// TIA Portal V20 export
ORGANIZATION_BLOCK "Startup"   // OB1050, LAD, Startup
TITLE = "Complete Restart"
AUTHOR : ERsystem_FA2_DH. Kim
// stored: AutoNumber false, IsIECCheckEnabled true, Namespace Unit1.Em5, SetENOAutomatically false
   VAR_INPUT
      LostRetentive : Bool;   // True if retentive data are lost
      LostRTC : Bool;   // True if date and time are lost
   END_VAR
BEGIN

REGION Network 1 (SCL): Build the Absolut Reference Designator
   // Set the Absoult Reference Designator in the Config DB
   IF LEN(IN := "Unit1.Em5.Config".em.referenceDesignator.parent) <> 0 THEN
     "Unit1.Em5.Config".em.referenceDesignator.combined := CONCAT_WSTRING(IN1 := "Unit1.Em5.Config".em.referenceDesignator.parent, IN2 := WSTRING#'.', IN3 := "Unit1.Em5.Config".em.referenceDesignator.relative);
   ELSE
     "Unit1.Em5.Config".em.referenceDesignator.combined := "Unit1.Em5.Config".em.referenceDesignator.relative;
   END_IF;
END_REGION

REGION Network 2 (SCL): Assign axes data
   //Assign axes
   "Unit1.Em5.Config".axis[1] := "BA040AZSCDR7_CathodeMainPnp1AxisX";
   "Unit1.Em5.Config".axis[2] := "BA040AZSCDR8_CathodeMainPnp2AxisX";
   "Unit1.Em5.Config".axis[3] := "BA040AZSCDR9_CathodeMainPnp1AxisY";
   "Unit1.Em5.Config".axis[4] := "BA040AZSCDR10_CathodeMainPnp1AxisZ";
   "Unit1.Em5.Config".axis[5] := "BA040AZSCDR13_CathodeMainPnp2AxisZ";
   "Unit1.Em5.Config".axis[6] := "BA040AZSCDR18_CathodeAlignTableAxisX";
   "Unit1.Em5.Config".axis[7] := "BA040AZSCDR19_CathodeAlignTableAxisY1";
   "Unit1.Em5.Config".axis[8] := "BA040AZSCDR20_CathodeAlignTableAxisY2";

   // Config.cam[1] := _.BA030AZSCDR5_cathodeMainPnp1AxisXCamMain;
   // Config.cam[2] := _.BA030AZSCDR6_cathodeMainPnp2AxisXCamMain;
   // Config.cam[3] := _.BA030AZSCDR12_cathodeMainPnp1AxisZCamMain;
   // Config.cam[4] := _.BA030AZSCDR14_cathodeMainPnp2AxisZCamMain;

   "Unit1.Em5.Config".outputCam[1] := "CathodePnP1XFwd";
   "Unit1.Em5.Config".outputCam[2] := "CathodePnP1XBwd";
   "Unit1.Em5.Config".outputCam[3] := "CathodePnP2XFwd";
   "Unit1.Em5.Config".outputCam[4] := "CathodePnP2XBwd";
   "Unit1.Em5.Config".outputCam[5] := "CathodePnPZ1Down1";
   "Unit1.Em5.Config".outputCam[6] := "CathodePnPZ1Up1";
   "Unit1.Em5.Config".outputCam[7] := "CathodePnPZ2Down1";
   "Unit1.Em5.Config".outputCam[8] := "CathodePnPZ2Up1";
   "Unit1.Em5.Config".outputCam[9] := "CathodePnPZ1Down2";
   "Unit1.Em5.Config".outputCam[10] := "CathodePnPZ1Up2";
   "Unit1.Em5.Config".outputCam[11] := "CathodePnPZ2Down2";
   "Unit1.Em5.Config".outputCam[12] := "CathodePnPZ2Up2";
   "Unit1.Em5.Config".outputCam[13] := "CathodePnPZ1SuctionOn";
   "Unit1.Em5.Config".outputCam[14] := "CathodePnPZ1SuctionOff";
   "Unit1.Em5.Config".outputCam[15] := "CathodePnPZ1ReelCutBlow";
   "Unit1.Em5.Config".outputCam[16] := "CathodePnPZ2SuctionOn";
   "Unit1.Em5.Config".outputCam[17] := "CathodePnPZ2SuctionOff";
   "Unit1.Em5.Config".outputCam[18] := "CathodeAlignSuctionOn";
   "Unit1.Em5.Config".outputCam[19] := "CathodeAlignSuctionOff";

   // Assign configuration data of axis

   // FB Enable
   "Unit1.Em5.HmiInterface".cmCathodeMainPnP1AxisX.commands.enableMasterControl := TRUE;
   "Unit1.Em5.HmiInterface".cmCathodeMainPnP1AxisY.commands.enableMasterControl := TRUE;
   "Unit1.Em5.HmiInterface".cmCathodeMainPnP1AxisZ.commands.enableMasterControl := TRUE;
   "Unit1.Em5.HmiInterface".cmCathodeMainPnP2AxisX.commands.enableMasterControl := TRUE;
   "Unit1.Em5.HmiInterface".cmCathodeMainPnP2AxisZ.commands.enableMasterControl := TRUE;
   "Unit1.Em5.HmiInterface".cmCathodeAlignTableAxisX.commands.enableMasterControl := TRUE;
   "Unit1.Em5.HmiInterface".cmCathodeAlignTableAxisY1.commands.enableMasterControl := TRUE;
   "Unit1.Em5.HmiInterface".cmCathodeAlignTableAxisY2.commands.enableMasterControl := TRUE;

   // Axis 1 BA030AZSCDR6_CathodeMainPnp1AxisX
   "Unit1.Em5.HmiInterface".cmCathodeMainPnP1AxisX.commandConfiguration.jog.velocity := 10.0;
   "Unit1.Em5.HmiInterface".cmCathodeMainPnP1AxisX.commandConfiguration.jog.acceleration := 100.0;
   "Unit1.Em5.HmiInterface".cmCathodeMainPnP1AxisX.commandConfiguration.jog.deceleration := 100.0;
   "Unit1.Em5.HmiInterface".cmCathodeMainPnP1AxisX.commandConfiguration.moveVelocity.velocity := 10.0;
   "Unit1.Em5.HmiInterface".cmCathodeMainPnP1AxisX.commandConfiguration.moveVelocity.acceleration := 100.0;
   "Unit1.Em5.HmiInterface".cmCathodeMainPnP1AxisX.commandConfiguration.moveVelocity.deceleration := 100.0;
   "Unit1.Em5.HmiInterface".cmCathodeMainPnP1AxisX.commandConfiguration.posRelative.velocity := 10.0;
   "Unit1.Em5.HmiInterface".cmCathodeMainPnP1AxisX.commandConfiguration.posRelative.acceleration := 100.0;
   "Unit1.Em5.HmiInterface".cmCathodeMainPnP1AxisX.commandConfiguration.posRelative.deceleration := 100.0;
   "Unit1.Em5.HmiInterface".cmCathodeMainPnP1AxisX.configuration.setPositions[0].name := 'reelCutConveyerPos';
   "Unit1.Em5.HmiInterface".cmCathodeMainPnP1AxisX.configuration.setPositions[1].name := 'alignTablePos';

   // Axis 2 BA030AZSCDR8_CathodeMainPnp2AxisX
   "Unit1.Em5.HmiInterface".cmCathodeMainPnP2AxisX.commandConfiguration.jog.velocity := 10.0;
   "Unit1.Em5.HmiInterface".cmCathodeMainPnP2AxisX.commandConfiguration.jog.acceleration := 100.0;
   "Unit1.Em5.HmiInterface".cmCathodeMainPnP2AxisX.commandConfiguration.jog.deceleration := 100.0;
   "Unit1.Em5.HmiInterface".cmCathodeMainPnP2AxisX.commandConfiguration.moveVelocity.velocity := 10.0;
   "Unit1.Em5.HmiInterface".cmCathodeMainPnP2AxisX.commandConfiguration.moveVelocity.acceleration := 100.0;
   "Unit1.Em5.HmiInterface".cmCathodeMainPnP2AxisX.commandConfiguration.moveVelocity.deceleration := 100.0;
   "Unit1.Em5.HmiInterface".cmCathodeMainPnP2AxisX.commandConfiguration.posRelative.velocity := 10.0;
   "Unit1.Em5.HmiInterface".cmCathodeMainPnP2AxisX.commandConfiguration.posRelative.acceleration := 100.0;
   "Unit1.Em5.HmiInterface".cmCathodeMainPnP2AxisX.commandConfiguration.posRelative.deceleration := 100.0;
   "Unit1.Em5.HmiInterface".cmCathodeMainPnP2AxisX.configuration.setPositions[0].name := 'alignTablePos';
   "Unit1.Em5.HmiInterface".cmCathodeMainPnP2AxisX.configuration.setPositions[1].name := 'stackTablePos';

   // Axis3 BA030AZSCDR11_CathodeMainPnp1AxisY
   "Unit1.Em5.HmiInterface".cmCathodeMainPnP1AxisY.commandConfiguration.jog.velocity := 10.0;
   "Unit1.Em5.HmiInterface".cmCathodeMainPnP1AxisY.commandConfiguration.jog.acceleration := 100.0;
   "Unit1.Em5.HmiInterface".cmCathodeMainPnP1AxisY.commandConfiguration.jog.deceleration := 100.0;
   "Unit1.Em5.HmiInterface".cmCathodeMainPnP1AxisY.commandConfiguration.moveVelocity.velocity := 10.0;
   "Unit1.Em5.HmiInterface".cmCathodeMainPnP1AxisY.commandConfiguration.moveVelocity.acceleration := 100.0;
   "Unit1.Em5.HmiInterface".cmCathodeMainPnP1AxisY.commandConfiguration.moveVelocity.deceleration := 100.0;
   "Unit1.Em5.HmiInterface".cmCathodeMainPnP1AxisY.commandConfiguration.posRelative.velocity := 10.0;
   "Unit1.Em5.HmiInterface".cmCathodeMainPnP1AxisY.commandConfiguration.posRelative.acceleration := 100.0;
   "Unit1.Em5.HmiInterface".cmCathodeMainPnP1AxisY.commandConfiguration.posRelative.deceleration := 100.0;
   "Unit1.Em5.HmiInterface".cmCathodeMainPnP1AxisY.configuration.setPositions[0].name := 'waitPos';

   // Axis 4 BA030AZSCDR12_CathodeMainPnp1AxisZ
   "Unit1.Em5.HmiInterface".cmCathodeMainPnP1AxisZ.commandConfiguration.jog.velocity := 10.0;
   "Unit1.Em5.HmiInterface".cmCathodeMainPnP1AxisZ.commandConfiguration.jog.acceleration := 100.0;
   "Unit1.Em5.HmiInterface".cmCathodeMainPnP1AxisZ.commandConfiguration.jog.deceleration := 100.0;
   "Unit1.Em5.HmiInterface".cmCathodeMainPnP1AxisZ.commandConfiguration.moveVelocity.velocity := 10.0;
   "Unit1.Em5.HmiInterface".cmCathodeMainPnP1AxisZ.commandConfiguration.moveVelocity.acceleration := 100.0;
   "Unit1.Em5.HmiInterface".cmCathodeMainPnP1AxisZ.commandConfiguration.moveVelocity.deceleration := 100.0;
   "Unit1.Em5.HmiInterface".cmCathodeMainPnP1AxisZ.commandConfiguration.posRelative.velocity := 10.0;
   "Unit1.Em5.HmiInterface".cmCathodeMainPnP1AxisZ.commandConfiguration.posRelative.acceleration := 100.0;
   "Unit1.Em5.HmiInterface".cmCathodeMainPnP1AxisZ.commandConfiguration.posRelative.deceleration := 100.0;
   "Unit1.Em5.HmiInterface".cmCathodeMainPnP1AxisZ.configuration.setPositions[0].name := 'upPos';
   "Unit1.Em5.HmiInterface".cmCathodeMainPnP1AxisZ.configuration.setPositions[1].name := 'reelCutConveyerDownPos';
   "Unit1.Em5.HmiInterface".cmCathodeMainPnP1AxisZ.configuration.setPositions[2].name := 'ailgnTableDownPos';

   // Axis 5 BA030AZSCDR14_CathodeMainPnp2AxisZ
   "Unit1.Em5.HmiInterface".cmCathodeMainPnP2AxisZ.commandConfiguration.jog.velocity := 10.0;
   "Unit1.Em5.HmiInterface".cmCathodeMainPnP2AxisZ.commandConfiguration.jog.acceleration := 100.0;
   "Unit1.Em5.HmiInterface".cmCathodeMainPnP2AxisZ.commandConfiguration.jog.deceleration := 100.0;
   "Unit1.Em5.HmiInterface".cmCathodeMainPnP2AxisZ.commandConfiguration.moveVelocity.velocity := 10.0;
   "Unit1.Em5.HmiInterface".cmCathodeMainPnP2AxisZ.commandConfiguration.moveVelocity.acceleration := 100.0;
   "Unit1.Em5.HmiInterface".cmCathodeMainPnP2AxisZ.commandConfiguration.moveVelocity.deceleration := 100.0;
   "Unit1.Em5.HmiInterface".cmCathodeMainPnP2AxisZ.commandConfiguration.posRelative.velocity := 10.0;
   "Unit1.Em5.HmiInterface".cmCathodeMainPnP2AxisZ.commandConfiguration.posRelative.acceleration := 100.0;
   "Unit1.Em5.HmiInterface".cmCathodeMainPnP2AxisZ.commandConfiguration.posRelative.deceleration := 100.0;
   "Unit1.Em5.HmiInterface".cmCathodeMainPnP2AxisZ.configuration.setPositions[0].name := 'upPos';
   "Unit1.Em5.HmiInterface".cmCathodeMainPnP2AxisZ.configuration.setPositions[1].name := 'ailgnTableDownPos';
   "Unit1.Em5.HmiInterface".cmCathodeMainPnP2AxisZ.configuration.setPositions[2].name := 'stackTableDownPos';

   // Axis 6 BA030AZSCDR18_CathodeAlignTableAxisX
   "Unit1.Em5.HmiInterface".cmCathodeAlignTableAxisX.commandConfiguration.jog.velocity := 10.0;
   "Unit1.Em5.HmiInterface".cmCathodeAlignTableAxisX.commandConfiguration.jog.acceleration := 100.0;
   "Unit1.Em5.HmiInterface".cmCathodeAlignTableAxisX.commandConfiguration.jog.deceleration := 100.0;
   "Unit1.Em5.HmiInterface".cmCathodeAlignTableAxisX.commandConfiguration.moveVelocity.velocity := 10.0;
   "Unit1.Em5.HmiInterface".cmCathodeAlignTableAxisX.commandConfiguration.moveVelocity.acceleration := 100.0;
   "Unit1.Em5.HmiInterface".cmCathodeAlignTableAxisX.commandConfiguration.moveVelocity.deceleration := 100.0;
   "Unit1.Em5.HmiInterface".cmCathodeAlignTableAxisX.commandConfiguration.posRelative.velocity := 10.0;
   "Unit1.Em5.HmiInterface".cmCathodeAlignTableAxisX.commandConfiguration.posRelative.acceleration := 100.0;
   "Unit1.Em5.HmiInterface".cmCathodeAlignTableAxisX.commandConfiguration.posRelative.deceleration := 100.0;
   "Unit1.Em5.HmiInterface".cmCathodeAlignTableAxisX.configuration.setPositions[0].name := 'waitPos';
   "Unit1.Em5.HmiInterface".cmCathodeAlignTableAxisX.configuration.setPositions[1].name := 'adjustPos';

   // Axis 7 BA030AZSCDR19_CathodeAlignTableAxisY1
   "Unit1.Em5.HmiInterface".cmCathodeAlignTableAxisY1.commandConfiguration.jog.velocity := 10.0;
   "Unit1.Em5.HmiInterface".cmCathodeAlignTableAxisY1.commandConfiguration.jog.acceleration := 100.0;
   "Unit1.Em5.HmiInterface".cmCathodeAlignTableAxisY1.commandConfiguration.jog.deceleration := 100.0;
   "Unit1.Em5.HmiInterface".cmCathodeAlignTableAxisY1.commandConfiguration.moveVelocity.velocity := 10.0;
   "Unit1.Em5.HmiInterface".cmCathodeAlignTableAxisY1.commandConfiguration.moveVelocity.acceleration := 100.0;
   "Unit1.Em5.HmiInterface".cmCathodeAlignTableAxisY1.commandConfiguration.moveVelocity.deceleration := 100.0;
   "Unit1.Em5.HmiInterface".cmCathodeAlignTableAxisY1.commandConfiguration.posRelative.velocity := 10.0;
   "Unit1.Em5.HmiInterface".cmCathodeAlignTableAxisY1.commandConfiguration.posRelative.acceleration := 100.0;
   "Unit1.Em5.HmiInterface".cmCathodeAlignTableAxisY1.commandConfiguration.posRelative.deceleration := 100.0;
   "Unit1.Em5.HmiInterface".cmCathodeAlignTableAxisY1.configuration.setPositions[0].name := 'waitPos';
   "Unit1.Em5.HmiInterface".cmCathodeAlignTableAxisY1.configuration.setPositions[1].name := 'adjustPos';

   // Axis 8 BA030AZSCDR20_CathodeAlignTableAxisY2
   "Unit1.Em5.HmiInterface".cmCathodeAlignTableAxisY2.commandConfiguration.jog.velocity := 10.0;
   "Unit1.Em5.HmiInterface".cmCathodeAlignTableAxisY2.commandConfiguration.jog.acceleration := 100.0;
   "Unit1.Em5.HmiInterface".cmCathodeAlignTableAxisY2.commandConfiguration.jog.deceleration := 100.0;
   "Unit1.Em5.HmiInterface".cmCathodeAlignTableAxisY2.commandConfiguration.moveVelocity.velocity := 10.0;
   "Unit1.Em5.HmiInterface".cmCathodeAlignTableAxisY2.commandConfiguration.moveVelocity.acceleration := 100.0;
   "Unit1.Em5.HmiInterface".cmCathodeAlignTableAxisY2.commandConfiguration.moveVelocity.deceleration := 100.0;
   "Unit1.Em5.HmiInterface".cmCathodeAlignTableAxisY2.commandConfiguration.posRelative.velocity := 10.0;
   "Unit1.Em5.HmiInterface".cmCathodeAlignTableAxisY2.commandConfiguration.posRelative.acceleration := 100.0;
   "Unit1.Em5.HmiInterface".cmCathodeAlignTableAxisY2.commandConfiguration.posRelative.deceleration := 100.0;
   "Unit1.Em5.HmiInterface".cmCathodeAlignTableAxisY2.configuration.setPositions[0].name := 'waitPos';
   "Unit1.Em5.HmiInterface".cmCathodeAlignTableAxisY2.configuration.setPositions[1].name := 'adjustPos';
END_REGION

REGION Network 3 (SCL): Assign TwoWayActuator data
   //Assign Configuration data of TwoWayActuator

   //cmCathodeMainPnP1RotaryCwCcw
   "Unit1.Em5.Config".cmCathodeMainPnP1RotaryCwCcw.referenceDesignator := WSTRING#'MainPnP1RotaryCwCcw';
   "Unit1.Em5.Config".cmCathodeMainPnP1RotaryCwCcw.disableFeedbackHomePos := FALSE;
   "Unit1.Em5.Config".cmCathodeMainPnP1RotaryCwCcw.disableFeedbackWorkPos := FALSE;
   "Unit1.Em5.HmiInterface".cmCathodeMainPnP1RotaryCwCcw.configuration.referenceDesignator := WSTRING#'MainPnP1RotaryCwCcw';
   "Unit1.Em5.HmiInterface".cmCathodeMainPnP1RotaryCwCcw.configuration.disableFeedbackHomePos := FALSE;
   "Unit1.Em5.HmiInterface".cmCathodeMainPnP1RotaryCwCcw.configuration.disableFeedbackWorkPos := FALSE;

   //cmCathodeMainPnP1SuctionPlateVacuum
   "Unit1.Em5.Config".cmCathodeMainPnP1SuctionPlateVacuum.referenceDesignator := WSTRING#'MainPnP1Vacuum';
   "Unit1.Em5.Config".cmCathodeMainPnP1SuctionPlateVacuum.disableFeedbackHomePos := FALSE;
   "Unit1.Em5.Config".cmCathodeMainPnP1SuctionPlateVacuum.disableFeedbackWorkPos := FALSE;
   "Unit1.Em5.HmiInterface".cmCathodeMainPnP1SuctionPlateVacuum.configuration.referenceDesignator := WSTRING#'MainPnP1Vacuum';
   "Unit1.Em5.HmiInterface".cmCathodeMainPnP1SuctionPlateVacuum.configuration.disableFeedbackHomePos := FALSE;
   "Unit1.Em5.HmiInterface".cmCathodeMainPnP1SuctionPlateVacuum.configuration.disableFeedbackWorkPos := FALSE;

   //cmCathodeMainPnP2SuctionPlateVacuum
   "Unit1.Em5.Config".cmCathodeMainPnP2SuctionPlateVacuum.referenceDesignator := WSTRING#'MainPnP2Vacuum';
   "Unit1.Em5.Config".cmCathodeMainPnP2SuctionPlateVacuum.disableFeedbackHomePos := FALSE;
   "Unit1.Em5.Config".cmCathodeMainPnP2SuctionPlateVacuum.disableFeedbackWorkPos := FALSE;
   "Unit1.Em5.HmiInterface".cmCathodeMainPnP2SuctionPlateVacuum.configuration.referenceDesignator := WSTRING#'MainPnP2Vacuum';
   "Unit1.Em5.HmiInterface".cmCathodeMainPnP2SuctionPlateVacuum.configuration.disableFeedbackHomePos := FALSE;
   "Unit1.Em5.HmiInterface".cmCathodeMainPnP2SuctionPlateVacuum.configuration.disableFeedbackWorkPos := FALSE;

   //cmCathodeAlignTableSuctionPlateVacuum
   "Unit1.Em5.Config".cmCathodeAlignTableSuctionPlateVacuum.referenceDesignator := WSTRING#'AlignTableVaccum';
   "Unit1.Em5.Config".cmCathodeAlignTableSuctionPlateVacuum.disableFeedbackHomePos := FALSE;
   "Unit1.Em5.Config".cmCathodeAlignTableSuctionPlateVacuum.disableFeedbackWorkPos := FALSE;
   "Unit1.Em5.HmiInterface".cmCathodeAlignTableSuctionPlateVacuum.configuration.referenceDesignator := WSTRING#'AlignTableVaccum';
   "Unit1.Em5.HmiInterface".cmCathodeAlignTableSuctionPlateVacuum.configuration.disableFeedbackHomePos := FALSE;
   "Unit1.Em5.HmiInterface".cmCathodeAlignTableSuctionPlateVacuum.configuration.disableFeedbackWorkPos := FALSE;

   //cmCathodeGlassCleaning
   "Unit1.Em5.Config".cmCathodeGlassCleaning.referenceDesignator := WSTRING#'GlassCleaning';
   "Unit1.Em5.Config".cmCathodeGlassCleaning.disableFeedbackHomePos := TRUE;
   "Unit1.Em5.Config".cmCathodeGlassCleaning.disableFeedbackWorkPos := TRUE;
   "Unit1.Em5.HmiInterface".cmCathodeGlassCleaning.configuration.referenceDesignator := WSTRING#'GlassCleaning';
   "Unit1.Em5.HmiInterface".cmCathodeGlassCleaning.configuration.disableFeedbackHomePos := TRUE;
   "Unit1.Em5.HmiInterface".cmCathodeGlassCleaning.configuration.disableFeedbackWorkPos := TRUE;

   //cmCathodeNgPnpUpDown
   "Unit1.Em5.Config".cmCathodeNgPnpUpDown.referenceDesignator := WSTRING#'NgPnpUpDown';
   "Unit1.Em5.Config".cmCathodeNgPnpUpDown.disableFeedbackHomePos := FALSE;
   "Unit1.Em5.Config".cmCathodeNgPnpUpDown.disableFeedbackWorkPos := FALSE;
   "Unit1.Em5.HmiInterface".cmCathodeNgPnpUpDown.configuration.referenceDesignator := WSTRING#'NgPnpUpDown';
   "Unit1.Em5.HmiInterface".cmCathodeNgPnpUpDown.configuration.disableFeedbackHomePos := FALSE;
   "Unit1.Em5.HmiInterface".cmCathodeNgPnpUpDown.configuration.disableFeedbackWorkPos := FALSE;

   //cmCathodeNgPnp1stFwdBwd
   "Unit1.Em5.Config".cmCathodeNgPnp1stFwdBwd.referenceDesignator := WSTRING#'NgPnp1stFwdBwd';
   "Unit1.Em5.Config".cmCathodeNgPnp1stFwdBwd.disableFeedbackHomePos := FALSE;
   "Unit1.Em5.Config".cmCathodeNgPnp1stFwdBwd.disableFeedbackWorkPos := FALSE;
   "Unit1.Em5.HmiInterface".cmCathodeNgPnp1stFwdBwd.configuration.referenceDesignator := WSTRING#'NgPnp1stFwdBwd';
   "Unit1.Em5.HmiInterface".cmCathodeNgPnp1stFwdBwd.configuration.disableFeedbackHomePos := FALSE;
   "Unit1.Em5.HmiInterface".cmCathodeNgPnp1stFwdBwd.configuration.disableFeedbackWorkPos := FALSE;

   //cmCathodeNgPnp2ndFwdBwd
   "Unit1.Em5.Config".cmCathodeNgPnp2ndFwdBwd.referenceDesignator := WSTRING#'NgPnp2ndFwdBwd';
   "Unit1.Em5.Config".cmCathodeNgPnp2ndFwdBwd.disableFeedbackHomePos := FALSE;
   "Unit1.Em5.Config".cmCathodeNgPnp2ndFwdBwd.disableFeedbackWorkPos := FALSE;
   "Unit1.Em5.HmiInterface".cmCathodeNgPnp2ndFwdBwd.configuration.referenceDesignator := WSTRING#'NgPnp2ndFwdBwd';
   "Unit1.Em5.HmiInterface".cmCathodeNgPnp2ndFwdBwd.configuration.disableFeedbackHomePos := FALSE;
   "Unit1.Em5.HmiInterface".cmCathodeNgPnp2ndFwdBwd.configuration.disableFeedbackWorkPos := FALSE;

   //cmCathodeMaintenanceMovingFixFrontRearFwdBwd
   "Unit1.Em5.Config".cmCathodeMaintenanceMovingFixFrontRearFwdBwd.referenceDesignator := WSTRING#'MaintenanceFix';
   "Unit1.Em5.Config".cmCathodeMaintenanceMovingFixFrontRearFwdBwd.disableFeedbackHomePos := FALSE;
   "Unit1.Em5.Config".cmCathodeMaintenanceMovingFixFrontRearFwdBwd.disableFeedbackWorkPos := FALSE;
   "Unit1.Em5.HmiInterface".cmCathodeMaintenanceMovingFixFrontRearFwdBwd.configuration.referenceDesignator := WSTRING#'MaintenanceFix';
   "Unit1.Em5.HmiInterface".cmCathodeMaintenanceMovingFixFrontRearFwdBwd.configuration.disableFeedbackHomePos := FALSE;
   "Unit1.Em5.HmiInterface".cmCathodeMaintenanceMovingFixFrontRearFwdBwd.configuration.disableFeedbackWorkPos := FALSE;

   //cmCathodeNgBoxLiftUpDown
   "Unit1.Em5.Config".cmCathodeNgBoxLiftUpDown.referenceDesignator := WSTRING#'NgBoxLiftUpDown';
   "Unit1.Em5.Config".cmCathodeNgBoxLiftUpDown.disableFeedbackHomePos := FALSE;
   "Unit1.Em5.Config".cmCathodeNgBoxLiftUpDown.disableFeedbackWorkPos := FALSE;
   "Unit1.Em5.HmiInterface".cmCathodeNgBoxLiftUpDown.configuration.referenceDesignator := WSTRING#'NgBoxLiftUpDown';
   "Unit1.Em5.HmiInterface".cmCathodeNgBoxLiftUpDown.configuration.disableFeedbackHomePos := FALSE;
   "Unit1.Em5.HmiInterface".cmCathodeNgBoxLiftUpDown.configuration.disableFeedbackWorkPos := FALSE;

   //cmCathodeNgBoxLockUpDown
   "Unit1.Em5.Config".cmCathodeNgBoxLockUpDown.referenceDesignator := WSTRING#'NgBoxLockUpDown';
   "Unit1.Em5.Config".cmCathodeNgBoxLockUpDown.disableFeedbackHomePos := FALSE;
   "Unit1.Em5.Config".cmCathodeNgBoxLockUpDown.disableFeedbackWorkPos := FALSE;
   "Unit1.Em5.HmiInterface".cmCathodeNgBoxLockUpDown.configuration.referenceDesignator := WSTRING#'NgBoxLockUpDown';
   "Unit1.Em5.HmiInterface".cmCathodeNgBoxLockUpDown.configuration.disableFeedbackHomePos := FALSE;
   "Unit1.Em5.HmiInterface".cmCathodeNgBoxLockUpDown.configuration.disableFeedbackWorkPos := FALSE;

   //cmCathodeNgPnpVaccum
   "Unit1.Em5.Config".cmCathodeNgPnpVaccum.referenceDesignator := WSTRING#'NgPnpVaccum';
   "Unit1.Em5.Config".cmCathodeNgPnpVaccum.disableFeedbackHomePos := FALSE;
   "Unit1.Em5.Config".cmCathodeNgPnpVaccum.disableFeedbackWorkPos := FALSE;
   "Unit1.Em5.HmiInterface".cmCathodeNgPnpVaccum.configuration.referenceDesignator := WSTRING#'NgPnpVaccum';
   "Unit1.Em5.HmiInterface".cmCathodeNgPnpVaccum.configuration.disableFeedbackHomePos := FALSE;
   "Unit1.Em5.HmiInterface".cmCathodeNgPnpVaccum.configuration.disableFeedbackWorkPos := FALSE;

   //cmCathodeConveyorCoverFwdBwd
   "Unit1.Em5.Config".cmCathodeConveyorCoverFwdBwd.referenceDesignator := WSTRING#'ConveyorCoverFwdBwd';
   "Unit1.Em5.Config".cmCathodeConveyorCoverFwdBwd.disableFeedbackHomePos := FALSE;
   "Unit1.Em5.Config".cmCathodeConveyorCoverFwdBwd.disableFeedbackWorkPos := FALSE;
   "Unit1.Em5.HmiInterface".cmCathodeConveyorCoverFwdBwd.configuration.referenceDesignator := WSTRING#'ConveyorCoverFwdBwd';
   "Unit1.Em5.HmiInterface".cmCathodeConveyorCoverFwdBwd.configuration.disableFeedbackHomePos := FALSE;
   "Unit1.Em5.HmiInterface".cmCathodeConveyorCoverFwdBwd.configuration.disableFeedbackWorkPos := FALSE;

   //cmCathodeConveyorPickUpBlower
   "Unit1.Em5.Config".cmCathodeConveyorPickUpBlower.referenceDesignator := WSTRING#'ConveyorPickUpBlower';
   "Unit1.Em5.Config".cmCathodeConveyorPickUpBlower.disableFeedbackHomePos := TRUE;
   "Unit1.Em5.Config".cmCathodeConveyorPickUpBlower.disableFeedbackWorkPos := TRUE;
   "Unit1.Em5.HmiInterface".cmCathodeConveyorPickUpBlower.configuration.referenceDesignator := WSTRING#'ConveyorPickUpBlower';
   "Unit1.Em5.HmiInterface".cmCathodeConveyorPickUpBlower.configuration.disableFeedbackHomePos := TRUE;
   "Unit1.Em5.HmiInterface".cmCathodeConveyorPickUpBlower.configuration.disableFeedbackWorkPos := TRUE;
END_REGION
END_ORGANIZATION_BLOCK
